// TIA Portal V18 export
DATA_BLOCK "Material Data current pgm"   // DB330
{ S7_Optimized_Access := 'TRUE' }
VERSION : 0.1
// stored: AutoNumber true, DBAccessibleFromOPCUA true, IsOnlyStoredInLoadMemory false, IsRetainMemResEnabled false, IsWriteProtectedInAS false, MemoryReserve 100
   VAR RETAIN
      Density : Struct
         "A" : Real;
         "B" : Real;
      END_STRUCT;
      Viscosity : Struct
         "A" : Real;
         "B" : Real;
      END_STRUCT;
      "Name" : Struct
         "A" : String[20];
         "B" : String[20];
      END_STRUCT;
      "name A+B" : String[40];
      "Mixed Density" : Real;
      BatchA : String[20];
      BatchB : String[20];
      "+symbol" : String := '+';
   END_VAR
BEGIN
END_DATA_BLOCK
